FUNCTION_BLOCK VECTOR_MULT_BY_SCALAR (* Multiply vector by scalar *)
  (* Standard: 61499-2 *)
  (* Version 1.0, 02-05-12, GASR, Universidade do Estado de Santa Catarina *)
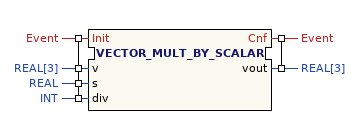
  EVENT_INPUT
    Init WITH v, s, div;
  END_EVENT
  EVENT_OUTPUT
    Cnf WITH vout;
  END_EVENT
  VAR_INPUT
    v : ARRAY [0..2] OF REAL;
    s : REAL;
    div : INT := 0;
  END_VAR
  VAR_OUTPUT
    vout : ARRAY [0..2] OF REAL;
  END_VAR
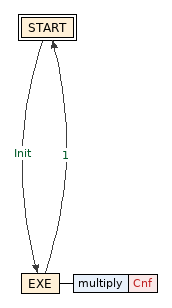
  EC_STATES
    START;
    EXE : multiply -> Cnf;
  END_STATES
  EC_TRANSITIONS
    START TO EXE := Init;
    EXE TO START := 1;
  END_TRANSITIONS
  ALGORITHM multiply IN Lua:
if( div == 1 ) then s = 1/s end
vout[1] = s*v[1]
vout[2] = s*v[2]
vout[3] = s*v[3]
  END_ALGORITHM
END_FUNCTION_BLOCK
